FUNCTION_BLOCK CHECK_POS (* Composite Function Block Type *)
  (* Standard: 61499-2 *)
  (* Version 0.2, 2003-12-05, JHC, Rockwell Automation, Renamed from NEWCOMPFB. *)
  (* Version 0.1, 2002-01-08, JHC, Rockwell Automation, Added DLY FB as example. *)
  (* Version 0.0, 2000-05-27, JHC, Rockwell Automation *)
  (* Compiler header: package fb.rt.template; *)
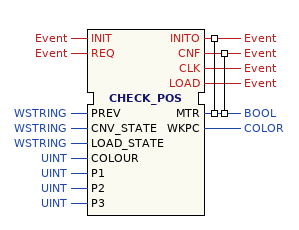
  EVENT_INPUT
    INIT; (* Initialization Request *)
    REQ; (* Normal Execution Request *)
  END_EVENT
  EVENT_OUTPUT
    INITO WITH MTR; (* Initialization Confirm *)
    CNF WITH MTR; (* Execution Confirmation *)
    CLK;
    LOAD;
  END_EVENT
  VAR_INPUT
    PREV : WSTRING;
    CNV_STATE : WSTRING;
    LOAD_STATE : WSTRING;
    COLOUR : UINT;
    P1 : UINT;
    P2 : UINT;
    P3 : UINT;
  END_VAR
  VAR_OUTPUT
    MTR : BOOL; (* Output event qualifier *)
    WKPC : COLOR;
  END_VAR
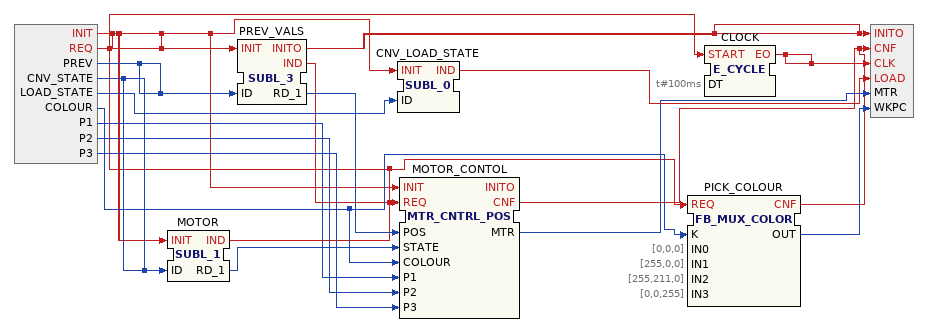
  FBS
    PREV_VALS : SUBL_3;
    MOTOR : SUBL_1;
    CNV_LOAD_STATE : SUBL_0;
    CLOCK : E_CYCLE(DT := t#100ms);
    MOTOR_CONTOL : MTR_CNTRL_POS;
    PICK_COLOUR : FB_MUX_COLOR(IN0 := [0,0,0], IN1 := [255,0,0], IN2 := [255,211,0], IN3 := [0,0,255]);
  END_FBS
  EVENT_CONNECTIONS
    INIT TO PREV_VALS.INIT;
    INIT TO MOTOR.INIT;
    INIT TO CNV_LOAD_STATE.INIT;
    CLOCK.EO TO CLK;
    REQ TO CLOCK.START;
    CNV_LOAD_STATE.IND TO LOAD;
    PREV_VALS.INITO TO INITO;
    INIT TO PREV_VALS.INIT;
    INIT TO MOTOR.INIT;
    INIT TO CNV_LOAD_STATE.INIT;
    CLOCK.EO TO CLK;
    REQ TO CLOCK.START;
    CNV_LOAD_STATE.IND TO LOAD;
    PREV_VALS.INITO TO INITO;
    INIT TO MOTOR_CONTOL.INIT;
    MOTOR_CONTOL.CNF TO CNF;
    REQ TO PICK_COLOUR.REQ;
    PICK_COLOUR.CNF TO CNF;
    PREV_VALS.IND TO MOTOR_CONTOL.REQ;
    REQ TO MOTOR_CONTOL.REQ;
    MOTOR.IND TO MOTOR_CONTOL.REQ;
  END_CONNECTIONS
  DATA_CONNECTIONS
    PREV TO PREV_VALS.ID;
    LOAD_STATE TO CNV_LOAD_STATE.ID;
    CNV_STATE TO MOTOR.ID;
    PREV TO PREV_VALS.ID;
    LOAD_STATE TO CNV_LOAD_STATE.ID;
    CNV_STATE TO MOTOR.ID;
    PREV_VALS.RD_1 TO MOTOR_CONTOL.POS;
    MOTOR.RD_1 TO MOTOR_CONTOL.STATE;
    COLOUR TO MOTOR_CONTOL.COLOUR;
    P1 TO MOTOR_CONTOL.P1;
    P2 TO MOTOR_CONTOL.P2;
    P3 TO MOTOR_CONTOL.P3;
    MOTOR_CONTOL.MTR TO MTR;
    COLOUR TO PICK_COLOUR.K;
    PICK_COLOUR.OUT TO WKPC;
  END_CONNECTIONS
END_FUNCTION_BLOCK
